(*************************************************************************************2.4Öá¹âÕ¤³ßÎ»ÖÃ¡¢ËÙ¶È¶Ô±È¼ì²é**********************************************************************)
IF  st_Power<>0 THEN
CASE moni_State OF
(*Top Î»ÖÃºÍËÙ¶È±È¶Ô*)
0:
		//实际(*Position*)
		(*Top*)
		Diff_UserTopPos_actual:=ABS(Pos_leftTopLin-Pos_RightTopLin);
		(*Bottom*)
		Diff_UserBottomPos_actual:=ABS(Pos_LeftBottomLin-Pos_RightBottomLin);
		(*Left*)
		Diff_UserLeftPos_actual:=ABS(Pos_LeftTopLin-Pos_LeftBottomLin);
		(*Right*)
		Diff_UserRightPos_actual:=ABS(Pos_RightTopLin-Pos_RightBottomLin);
		(*Velocity*)
		(*Top*)
		Diff_UserTopVelo_actual:=ABS(Velo_leftTopLin-Velo_RightTopLin);
		(*Bottom*)
		Diff_UserBottomVelo_actual:=ABS(Velo_LeftBottomLin-Velo_RightBottomLin);
		(*Left*)
		Diff_UserLeftVelo_actual:=ABS(Velo_LeftTopLin-Velo_LeftBottomLin);
		(*Right*)
		Diff_UserRightVelo_actual:=ABS(Velo_RightTopLin-Velo_RightBottomLin);
		//阈值
		Threshold_UserTopPos_PLC:=Threshold_UserTopPos+UserTaperPositionDisplay;//Top位置误差=gap运动细微误差+目标taper位置
		Threshold_UserTopVelo_PLC:=Threshold_UserTopVelo+ABS(UserGapVelocityDisplay);//Top速度误差=gap运动细微误差+gap目标速度。因为可能出现一个轴运动完了，另一个轴还在运动的情况
		Threshold_UserBottomPos_PLC:=Threshold_UserBottomPos+UserTaperPositionDisplay;//Bottom同上
		Threshold_UserBottomVelo_PLC:=Threshold_UserBottomVelo+ABS(UserGapVelocityDisplay);//Bottom同上
		Threshold_UserLeftPos_PLC:=Threshold_UserLeftPos+UserTaperPositionDisplay;
		Threshold_UserLeftVelo_PLC:=Threshold_UserLeftVelo+ABS(UserGapVelocityDisplay);
		Threshold_UserRightPos_PLC:=Threshold_UserRightPos+UserTaperPositionDisplay;
		Threshold_UserRightVelo_PLC:=Threshold_UserRightVelo+ABS(UserGapVelocityDisplay);
		//比较
		IF Diff_UserTopPos_actual >Threshold_UserTopPos_PLC THEN
				Error:=TRUE;
				ErrorID:=601;
				ErrorDescription:='Diff_UserTopPos_actual >Threshold_UserTopPos_PLC';
				moni_State:=-100;
		ELSIF Diff_UserTopVelo_actual>Threshold_UserTopVelo_PLC  THEN
				Error:=TRUE;
				ErrorID:=602;
				ErrorDescription:='Diff_UserTopVelo_actual>Threshold_UserTopVelo_PLC';
				moni_State:=-100;
		(*Bottom Î»ÖÃºÍËÙ¶È±È¶Ô*)
		ELSIF Diff_UserBottomPos_actual>Threshold_UserBottomPos_PLC THEN
				Error:=TRUE;
				ErrorID:=603;
				ErrorDescription:='Diff_UserBottomPos_actual>Threshold_UserBottomPos_PLC';
				moni_State:=-100;
		ELSIF Diff_UserBottomVelo_actual>Threshold_UserBottomVelo_PLC  THEN
				Error:=TRUE;
				ErrorID:=604;
				ErrorDescription:='Diff_UserBottomVelo_actual>Threshold_UserBottomVelo_PLC';
				moni_State:=-100;
		(*Left Î»ÖÃºÍËÙ¶È±È¶Ô*)
		ELSIF Diff_UserLeftPos_actual>Threshold_UserLeftPos_PLC  THEN
				Error:=TRUE;
				ErrorID:=605;
				ErrorDescription:='Diff_UserLeftPos_actual>Threshold_UserLeftPos_PLC';
				moni_State:=-100;
		ELSIF  Diff_UserLeftVelo_actual>Threshold_UserLeftVelo_PLC THEN
				Error:=TRUE;
				ErrorID:=606;
				ErrorDescription:='Diff_UserLeftVelo_actual>Threshold_UserLeftVelo_PLC';
				moni_State:=-100;
		(*Right Î»ÖÃºÍËÙ¶È±È¶Ô*)
		ELSIF Diff_UserRightPos_actual>Threshold_UserRightPos_PLC  THEN
				Error:=TRUE;
				ErrorID:=607;
				ErrorDescription:='Diff_UserRightPos_actual>Threshold_UserRightPos_PLC';
				moni_State:=-100;
		ELSIF  Diff_UserRightVelo_actual>Threshold_UserRightVelo_PLC THEN
				Error:=TRUE;
				ErrorID:=608;
				ErrorDescription:='Diff_UserRightVelo_actual>Threshold_UserRightVelo_PLC';
				moni_State:=-100;
		END_IF
-100:
		btn_UserGapStop:=TRUE;
		FB_PlcEmergencyStop();
		Error:=TRUE;
		LED_Error:=TRUE;
END_CASE
END_IF
END_ACTION

ACTION A_OneKeyToMaxGap:
//0.上升沿触发
//1.判断电机是否在开启状态,没有就打开电源
//2.判断是否在Moving状态,若有就Stop
//3.将磁间隙打开到至最大阈值
//4.到位后给出反馈
OneKeyToMaxGap_RTRIG(CLK:=btn_OneKeyToMaxGap);
IF OneKeyToMaxGap_RTRIG.Q THEN
	OneKeyToMaxGap_Triggered:=TRUE;
	OneKeyToMaxGap_Done:=FALSE;
END_IF
IF OneKeyToMaxGap_Triggered THEN
	CASE OneKeyToMaxGap_State OF
		0://1.判断电机是否在开启状态,没有就打开电源
			IF st_Power=1 THEN
				OneKeyToMaxGap_State:=1;
			ELSE
				btn_PowerOn:=TRUE;
				IF btn_PowerOn THEN
					A_PowerOn();
				END_IF
			END_IF
		1://1.判断是否在谱学扫描模式，如果是，则切换回正常运动模式
			IF IsSSMotionMode THEN
				SS_Stop:=TRUE;
				IsSSMotionMode:=FALSE;
			END_IF
			OneKeyToMaxGap_State:=2;
		2://判断是否在taper，如果在taper,则判断是否在运动，如果是，则停止运动,0.5sh后，转入下一步
			IF TaperOrNot THEN
				IF moveStatusLeftTop OR moveStatusRightTop OR moveStatusLeftBottom OR moveStatusRightBottom THEN
					btn_UserGapStop:=TRUE;
				ELSE
					OneKeyToMaxGap_TON_Stop2Move_InTaperMode(PT:=T#0.5S);
					OneKeyToMaxGap_TON_Stop2Move_InTaperMode.IN:=TRUE;
					IF OneKeyToMaxGap_TON_Stop2Move_InTaperMode.Q THEN
						TaperOrNot:=FALSE;//关闭taper模式
						OneKeyToMaxGap_State:=3;
						OneKeyToMaxGap_TON_Stop2Move_InTaperMode.IN:=FALSE;
					END_IF
				END_IF
			ELSE
				OneKeyToMaxGap_State:=3;
			END_IF
		3://3.判断是否在Moving状态,若有就Stop.Taper模式已处理完，此处开始走正常GAP开合逻辑
			IF moveStatusLeftTop OR moveStatusRightTop OR moveStatusLeftBottom OR moveStatusRightBottom THEN
				btn_UserGapStop:=TRUE;
			ELSE
				OneKeyToMaxGap_TON_Stop2Move(PT:=T#0.5S);
				OneKeyToMaxGap_TON_Stop2Move.IN:=TRUE;
				IF OneKeyToMaxGap_TON_Stop2Move.Q THEN
					OneKeyToMaxGap_State:=4;
					OneKeyToMaxGap_TON_Stop2Move.IN:=FALSE;
				END_IF
			END_IF
		4://4.将磁间隙打开到至最大阈值
			OneKeyToMaxGap_TON(PT:=INT_TO_TIME(LREAL_TO_INT(max_UserGapPositionNew+30))*1000);
			OneKeyToMaxGap_TON.IN:=TRUE;
			OneKeyToMaxGap_TON_Power2Move(PT:=T#0.1S);
			OneKeyToMaxGap_TON_Power2Move.IN:=TRUE;
			UserGapPositionNew:=max_UserGapPositionNew;
			UserGapVelocityNew:=1;
			btn_UserGapMove:=TRUE;
			IF OneKeyToMaxGap_TON_Power2Move.Q THEN
				OneKeyToMaxGap_TON_Power2Move.IN:=FALSE;
				IF FB_MOVE.BCGapDone THEN
					OneKeyToMaxGap_State:=88;
				END_IF
			END_IF
			IF OneKeyToMaxGap_TON.Q THEN//如果150s后，还没有运动到指定gap，则报错
				OneKeyToMaxGap_TON.IN:=FALSE;
				OneKeyToMaxGap_State:=-100;
			END_IF
		88://6.到位后给出反馈
			OneKeyToMaxGap_Done:=TRUE;	
			Error:=FALSE;
			ErrorID:=0;
			ErrorDescription:='';
			btn_OneKeyToMaxGap:=FALSE;
			OneKeyToMaxGap_Triggered:=FALSE;
			OneKeyToMaxGap_State:=0;
				
		-100:
			OneKeyToMaxGap_Done:=FALSE;
			Error:=TRUE;
			ErrorID:=1705;
			ErrorDescription:='OneKeyToMaxGap Fail';
			btn_OneKeyToMaxGap:=FALSE;
			OneKeyToMaxGap_Triggered:=FALSE;
			OneKeyToMaxGap_State:=0;
	END_CASE
END_IF
END_ACTION

ACTION A_PhaseLowerMotion:
(*输入保护*)
IF btn_UserPhaseLowerMove THEN
	IF NOT inRange_UserPhaseLowerPositionNew THEN
		btn_UserPhaseLowerStop:=TRUE;
		btn_UserPhaseLowerMove:=FALSE;
		Error:=TRUE;
		ErrorId:=812;
		ErrorDescription:='target PhaseLower position out of range,please check';
		RETURN;
	ELSE
		btn_UserPhaseLowerStop:=FALSE;
		Error:=FALSE;
		ErrorId:=0;
		ErrorDescription:='';	
	END_IF
	IF NOT inRange_UserPhaseLowerVelocityNew THEN
		btn_UserPhaseLowerStop:=TRUE;
		btn_UserPhaseLowerMove:=FALSE;
		Error:=TRUE;
		ErrorId:=813;
		ErrorDescription:='target PhaseLower velocity out of range,please check';
		RETURN;
	ELSE
		btn_UserPhaseLowerStop:=FALSE;
		Error:=FALSE;
		ErrorId:=0;
		ErrorDescription:='';
	END_IF
END_IF
(*改变Phase前，先检查Gap，Gap必须处于阈值之上（基本在最大间隙），才能改变Pase*)
IF GapPhase_ChainProtection_On AND UserGapPositionDisplay-GapPhase_ChainProtection_MaxGapValue<-0.01 AND btn_UserPhaseLowerMove THEN
		btn_UserPhaseLowerStop:=TRUE;
		btn_UserPhaseLowerMove:=FALSE;
		Error:=TRUE;
		ErrorId:=814;
		ErrorDescription:='Please Move Gap to MaxGapValue first before move Phase';
		RETURN;
END_IF

(*分别比较四轴目标位置与当前位置的差，如果目标位置比当前位置低，则需要运动到更低-回程差一半；再运动至最终目标位置*)
//只在m=和n=0的时候判断，否则会出现一些BUG，比如往大间隙开时，运动到位后m不能回到0.
IF m_state_PhaseLower=0 AND n_state_PhaseLower=0 THEN
	IF UserPhaseLowerPositionNew-Pos_PhaseLowerLin<-LEDriftErrorThreshold_PhaseLower THEN
			TargetPosLessThanCurrentPos_PhaseLower:=TRUE;
	ELSE
			TargetPosLessThanCurrentPos_PhaseLower:=FALSE;
	END_IF
END_IF

(*Move*)
IF InitPowerDone THEN
		(*目标位置都大于当前位置，直接走到目标位置即可，不需要先走到考虑回城误差的临时位置*)
		IF NOT TargetPosLessThanCurrentPos_PhaseLower AND NOT HysteresisMoving_PhaseLower THEN
			CASE m_state_PhaseLower OF
				0:
					FB_Move_PhaseLower.Mode:=4;						//1.gap;2.single;3.taper;4.debug;5.BCGap&UserMode
					FB_Move_PhaseLower.CoupleState:=st_Couple;			
					FB_Move_PhaseLower.PowerState:=st_Power;							
					FB_Move_PhaseLower.PhaseLowerPosition:=UserPhaseLowerPositionNew;
					FB_Move_PhaseLower.PhaseLowerVelocity:=UserPhaseLowerVelocityNew;		
					IF btn_UserPhaseLowerMove THEN
						FB_Move_PhaseLower.PhaseLowerMove:=TRUE;
						m_state_PhaseLower:=1;
						FB_Move_PhaseLower();
					END_IF
				1:
					btn_UserPhaseLowerMove:=FALSE;
					FB_Move_PhaseLower();
					IF NOT FB_Move_PhaseLower.PhaseLowerDone THEN			(*ÔË¶¯Î´Íê³É£¬Ñ­»·*)
						Led_Run:=TRUE;
						m_state_PhaseLower:=1;
					ELSE									(*ÔË¶¯Íê³É£¬ÏÂÒ»²½*)
						m_state_PhaseLower:=88;
					END_IF
				88:
					btn_UserPhaseLowerMove:=FALSE;					(*×´Ì¬»Ö¸´*)
					Led_Run:=FALSE;
					m_state_PhaseLower:=0;
			END_CASE
		(*四轴有目标位置小于当前位置，先走到临时位置，再走到目标位置*)
		ELSE
			CASE n_state_PhaseLower OF
				0:
					FB_Move_PhaseLower.Mode:=4;						//1.gap;2.single;3.taper;4.debug;5.BCGap&UserMode;5:userMode_2
					FB_Move_PhaseLower.CoupleState:=st_Couple;			
					FB_Move_PhaseLower.PowerState:=st_Power;			
					
					//
					IF TargetPosLessThanCurrentPos_PhaseLower THEN			
						FB_Move_PhaseLower.PhaseLowerPosition:=UserPhaseLowerPositionNew-HysteresisError_PhaseLower;
					ELSE
						FB_Move_PhaseLower.PhaseLowerPosition:=UserPhaseLowerPositionNew;	
					END_IF				
					//
					FB_Move_PhaseLower.PhaseLowerVelocity:=UserPhaseLowerVelocityNew;
						
					IF btn_UserPhaseLowerMove THEN							
						n_state_PhaseLower:=1;
						FB_Move_PhaseLower.PhaseLowerMove:=TRUE;
						FB_Move_PhaseLower();
						HysteresisMoving_PhaseLower:=TRUE;
					END_IF
				1:
					btn_UserPhaseLowerMove:=FALSE;
					FB_Move_PhaseLower();
					IF NOT FB_Move_PhaseLower.PhaseLowerDone THEN			(*还未运动到位置,运动过程中*)
						Led_Run:=TRUE;
						n_state_PhaseLower:=1;
					ELSE									
						n_state_PhaseLower:=2;							(*转到下一步，运动到最终位置*)
						FB_Move_PhaseLower.PhaseLowerMove:=FALSE;
						//Led_Run:=FALSE;
					END_IF
				2:
					FB_Move_PhaseLower.PhaseLowerReset:=FALSE;
					FB_Move_PhaseLower.Mode:=4;						//1.gap;2.single;3.taper;4.debug;5.BCGap&UserMode
					FB_Move_PhaseLower.CoupleState:=st_Couple;			
					FB_Move_PhaseLower.PowerState:=st_Power;			
					FB_Move_PhaseLower.PhaseLowerMove:=TRUE;
					//直接走到目标位置，已经走到位置的，可以继续下命令，只不过它不在走了而已
					FB_Move_PhaseLower.PhaseLowerPosition:=UserPhaseLowerPositionNew;	
					FB_Move_PhaseLower.PhaseLowerVelocity:=UserPhaseLowerVelocityNew;
					FB_Move_PhaseLower();							
					n_state_PhaseLower:=3;
				3:
					FB_Move_PhaseLower();
					IF NOT FB_Move_PhaseLower.PhaseLowerDone THEN			(*还未运动到位置,运动过程中*)
						Led_Run:=TRUE;
						n_state_PhaseLower:=3;
					ELSE									
						n_state_PhaseLower:=88;							(*运动到了最终位置*)
					END_IF
				88:
					btn_UserPhaseLowerMove:=FALSE;					
					Led_Run:=FALSE;
					n_state_PhaseLower:=0;
					HysteresisMoving_PhaseLower:=FALSE;
			END_CASE
		END_IF
	//END_IF
END_IF

IF btn_UserPhaseLowerStop THEN
	FB_Move_PhaseLower.PhaseLowerReset:=TRUE;							(*¸øÔË¶¯FB¸øÍ£Ö¹ÐÅºÅ£¬Ê¹FB_Move×´Ì¬»Ö¸´*)
	FB_Move_PhaseLower();											(*Æô¶¯FB_Move*)
	btn_UserPhaseLowerMove:=FALSE;								(*btn_GapMove:=FALSE*)
	m_state_PhaseLower:=0;	
	n_state_PhaseLower:=0;										(*m_state:=0;*)
	CASE s_state_PhaseLower OF
			0:
				FB_Stop_PhaseLower.Mode:=4;							(*1£ºgapÄ£Ê½£»2£ºµ¥ÁºÄ£Ê½£»3£ºtaperÄ£Ê½£»4£ºDebugÄ£Ê½£»5£ºBCGapÄ£Ê½*)
				FB_Stop_PhaseLower.CoupleState:=st_Couple;			(*ñîºÏ×´Ì¬ÊäÈë*)
				FB_Stop_PhaseLower.PowerState:=st_Power;				(*µçÔ´×´Ì¬ÊäÈë*)
				FB_Stop_PhaseLower.PhaseLowerStop:=TRUE;				(*Execute TRUE*)
				FB_Stop_PhaseLower();								(*Æô¶¯FB*)
				s_state_PhaseLower:=1;
			1:
				FB_Stop_PhaseLower();
				IF NOT FB_Stop_PhaseLower.PhaseLowerDone THEN			(*Í£Ö¹Î´Íê³É£¬Ñ­»·*)
					s_state_PhaseLower:=1;
				ELSE									(*Í£Ö¹Íê³É£¬ÏÂÒ»²½*)
					s_state_PhaseLower:=88;
				END_IF
			88:
				btn_UserPhaseLowerStop:=FALSE;						(*»Ö¸´×´Ì¬*)
				FB_Move_PhaseLower.PhaseLowerReset:=FALSE;				(*ÔËÐÐFB*)
				s_state_PhaseLower:=0;
		END_CASE
END_IF

(*触发限位开关后，相当于点击了Stop按钮*)
FTrig_ReachLS_PhaseLower(CLK:=LS_PhaseLower_Entrance AND LS_PhaseLower_Exit);
IF FTrig_ReachLS_PhaseLower.Q THEN
	btn_UserPhaseLowerStop:=TRUE;
END_IF
END_ACTION

ACTION A_PhaseUpperMotion:
(*输入保护*)
IF btn_UserPhaseUpperMove THEN
	IF NOT inRange_UserPhaseUpperPositionNew THEN
		btn_UserPhaseUpperStop:=TRUE;
		btn_UserPhaseUpperMove:=FALSE;
		Error:=TRUE;
		ErrorId:=809;
		ErrorDescription:='target PhaseUpper position out of range,please check';
		RETURN;
	ELSE
		btn_UserPhaseUpperStop:=FALSE;
		Error:=FALSE;
		ErrorId:=0;
		ErrorDescription:='';	
	END_IF
	IF NOT inRange_UserPhaseUpperVelocityNew THEN
		btn_UserPhaseUpperStop:=TRUE;
		btn_UserPhaseUpperMove:=FALSE;
		Error:=TRUE;
		ErrorId:=810;
		ErrorDescription:='target PhaseUpper velocity out of range,please check';
		RETURN;
	ELSE
		btn_UserPhaseUpperStop:=FALSE;
		Error:=FALSE;
		ErrorId:=0;
		ErrorDescription:='';
	END_IF
END_IF
(*改变Phase前，先检查Gap，Gap必须处于阈值之上（基本在最大间隙），才能改变Pase*)
IF GapPhase_ChainProtection_On AND UserGapPositionDisplay-GapPhase_ChainProtection_MaxGapValue<-0.01 AND btn_UserPhaseUpperMove THEN
		btn_UserPhaseUpperStop:=TRUE;
		btn_UserPhaseUpperMove:=FALSE;
		Error:=TRUE;
		ErrorId:=811;
		ErrorDescription:='Please Move Gap to MaxGapValue first before move Phase';
		RETURN;
END_IF
(*分别比较四轴目标位置与当前位置的差，如果目标位置比当前位置低，则需要运动到更低-回程差一半；再运动至最终目标位置*)
//只在m=和n=0的时候判断，否则会出现一些BUG，比如往大间隙开时，运动到位后m不能回到0.
IF m_state_PhaseUpper=0 AND n_state_PhaseUpper=0 THEN
	IF UserPhaseUpperPositionNew-Pos_PhaseUpperLin<-LEDriftErrorThreshold_PhaseUpper THEN
			TargetPosLessThanCurrentPos_PhaseUpper:=TRUE;
	ELSE
			TargetPosLessThanCurrentPos_PhaseUpper:=FALSE;
	END_IF
END_IF

(*Move*)
IF InitPowerDone THEN
		(*目标位置都大于当前位置，直接走到目标位置即可，不需要先走到考虑回城误差的临时位置*)
		IF NOT TargetPosLessThanCurrentPos_PhaseUpper AND NOT HysteresisMoving_PhaseUpper THEN
			CASE m_state_PhaseUpper OF
				0:
					FB_Move_PhaseUpper.Mode:=4;						//1.gap;2.single;3.taper;4.debug;5.BCGap&UserMode
					FB_Move_PhaseUpper.CoupleState:=st_Couple;			
					FB_Move_PhaseUpper.PowerState:=st_Power;	
					IF btn_UserPhaseUpperMove THEN						
						IF NOT st_Power THEN
							ErrorID:=1501;
							Error:=TRUE;
							ErrorDescription:='Plz PowerOn Frist';
							LED_Error:=TRUE;
							//btn_UserGapMove:=FALSE;
							RETURN;
						ELSE
							ErrorID:=0;
							Error:=FALSE;
							ErrorDescription:='';
							LED_Error:=FALSE;
							//btn_UserGapMove:=TRUE;
						END_IF
						//目标速度位置赋值
						FB_Move_PhaseUpper.PhaseUpperPosition:=UserPhaseUpperPositionNew;
						FB_Move_PhaseUpper.PhaseUpperVelocity:=UserPhaseUpperVelocityNew;		
						//Move
						FB_Move_PhaseUpper.PhaseUpperMove:=TRUE;
						m_state_PhaseUpper:=1;
						FB_Move_PhaseUpper();
					END_IF
				1:
					btn_UserPhaseUpperMove:=FALSE;
					FB_Move_PhaseUpper();
					IF NOT FB_Move_PhaseUpper.PhaseUpperDone THEN			(*ÔË¶¯Î´Íê³É£¬Ñ­»·*)
						Led_Run:=TRUE;
						m_state_PhaseUpper:=1;
					ELSE									(*ÔË¶¯Íê³É£¬ÏÂÒ»²½*)
						m_state_PhaseUpper:=88;
					END_IF
				88:
					btn_UserPhaseUpperMove:=FALSE;					(*×´Ì¬»Ö¸´*)
					Led_Run:=FALSE;
					m_state_PhaseUpper:=0;
			END_CASE
		(*四轴有目标位置小于当前位置，先走到临时位置，再走到目标位置*)
		ELSE
			CASE n_state_PhaseUpper OF
				0:
					FB_Move_PhaseUpper.Mode:=4;						//1.gap;2.single;3.taper;4.debug;5.BCGap&UserMode;5:userMode_2
					FB_Move_PhaseUpper.CoupleState:=st_Couple;			
					FB_Move_PhaseUpper.PowerState:=st_Power;			
					//
					IF btn_UserPhaseUpperMove THEN
						IF NOT st_Power THEN
							ErrorID:=1501;
							Error:=TRUE;
							ErrorDescription:='Plz PowerOn Frist';
							LED_Error:=TRUE;
							//btn_UserGapMove:=FALSE;
							RETURN;
						ELSE
							ErrorID:=0;
							Error:=FALSE;
							ErrorDescription:='';
							LED_Error:=FALSE;
							//btn_UserGapMove:=TRUE;	
						END_IF
						IF TargetPosLessThanCurrentPos_PhaseUpper THEN			
							FB_Move_PhaseUpper.PhaseUpperPosition:=UserPhaseUpperPositionNew-HysteresisError_PhaseUpper;
						ELSE
							FB_Move_PhaseUpper.PhaseUpperPosition:=UserPhaseUpperPositionNew;	
						END_IF				
						//	close gap情况下，加入了PositionNewTemp。//
						//如果在往小间隙运行过程中，改变了目标gap，会在第到达第一次目标位置后，继续向第二
						//次输入的目标运动，而不会回到第一次的目标位置。用temp锁定目标位置
						UserPhaseUpperPositionNewTemp:=UserPhaseUpperPositionNew;
						FB_Move_PhaseUpper.PhaseUpperVelocity:=UserPhaseUpperVelocityNew;
						
						FB_Move_PhaseUpper.PhaseUpperMove:=TRUE;
						FB_Move_PhaseUpper();
						HysteresisMoving_PhaseUpper:=TRUE;
						n_state_PhaseUpper:=1;
					END_IF
				1:
					btn_UserPhaseUpperMove:=FALSE;
					FB_Move_PhaseUpper();
					IF NOT FB_Move_PhaseUpper.PhaseUpperDone THEN			(*还未运动到位置,运动过程中*)
						Led_Run:=TRUE;
						n_state_PhaseUpper:=1;
					ELSE									
						n_state_PhaseUpper:=2;							(*转到下一步，运动到最终位置*)
						FB_Move_PhaseUpper.PhaseUpperMove:=FALSE;
						//Led_Run:=FALSE;
					END_IF
				2:
					FB_Move_PhaseUpper.PhaseUpperReset:=FALSE;
					FB_Move_PhaseUpper.Mode:=4;						//1.gap;2.single;3.taper;4.debug;5.BCGap&UserMode
					FB_Move_PhaseUpper.CoupleState:=st_Couple;			
					FB_Move_PhaseUpper.PowerState:=st_Power;			
					FB_Move_PhaseUpper.PhaseUpperMove:=TRUE;
					//直接走到目标位置，已经走到位置的，可以继续下命令，只不过它不在走了而已
					FB_Move_PhaseUpper.PhaseUpperPosition:=UserPhaseUpperPositionNewTemp;	
					FB_Move_PhaseUpper.PhaseUpperVelocity:=UserPhaseUpperVelocityNew;
					FB_Move_PhaseUpper();							
					n_state_PhaseUpper:=3;
				3:
					FB_Move_PhaseUpper();
					IF NOT FB_Move_PhaseUpper.PhaseUpperDone THEN			(*还未运动到位置,运动过程中*)
						Led_Run:=TRUE;
						n_state_PhaseUpper:=3;
					ELSE									
						n_state_PhaseUpper:=88;							(*运动到了最终位置*)
					END_IF
				88:
					btn_UserPhaseUpperMove:=FALSE;					
					Led_Run:=FALSE;
					n_state_PhaseUpper:=0;
					HysteresisMoving_PhaseUpper:=FALSE;
			END_CASE
		END_IF
	//END_IF
END_IF

IF btn_UserPhaseUpperStop THEN
	FB_Move_PhaseUpper.PhaseUpperReset:=TRUE;							(*¸øÔË¶¯FB¸øÍ£Ö¹ÐÅºÅ£¬Ê¹FB_Move×´Ì¬»Ö¸´*)
	FB_Move_PhaseUpper();											(*Æô¶¯FB_Move*)
	btn_UserPhaseUpperMove:=FALSE;								(*btn_GapMove:=FALSE*)
	m_state_PhaseUpper:=0;	
	n_state_PhaseUpper:=0;										(*m_state:=0;*)
	CASE s_state_PhaseUpper OF
			0:
				FB_Stop_PhaseUpper.Mode:=4;							(*1£ºgapÄ£Ê½£»2£ºµ¥ÁºÄ£Ê½£»3£ºtaperÄ£Ê½£»4£ºDebugÄ£Ê½£»5£ºBCGapÄ£Ê½*)
				FB_Stop_PhaseUpper.CoupleState:=st_Couple;			(*ñîºÏ×´Ì¬ÊäÈë*)
				FB_Stop_PhaseUpper.PowerState:=st_Power;				(*µçÔ´×´Ì¬ÊäÈë*)
				FB_Stop_PhaseUpper.PhaseUpperStop:=TRUE;				(*Execute TRUE*)
				FB_Stop_PhaseUpper();								(*Æô¶¯FB*)
				s_state_PhaseUpper:=1;
			1:
				FB_Stop_PhaseUpper();
				IF NOT FB_Stop_PhaseUpper.PhaseUpperDone THEN			(*Í£Ö¹Î´Íê³É£¬Ñ­»·*)
					s_state_PhaseUpper:=1;
				ELSE									(*Í£Ö¹Íê³É£¬ÏÂÒ»²½*)
					s_state_PhaseUpper:=88;
				END_IF
			88:
				btn_UserPhaseUpperStop:=FALSE;						(*»Ö¸´×´Ì¬*)
				FB_Move_PhaseUpper.PhaseUpperReset:=FALSE;				(*ÔËÐÐFB*)
				s_state_PhaseUpper:=0;
		END_CASE
END_IF

(*触发限位开关后，相当于点击了Stop按钮*)
FTrig_ReachLS_PhaseUpper(CLK:=LS_PhaseUpper_Entrance AND LS_PhaseUpper_Exit);
IF FTrig_ReachLS_PhaseUpper.Q THEN
	btn_UserPhaseUpperStop:=TRUE;
END_IF
END_ACTION

ACTION A_PowerOff:
CASE d_state OF
		0:(*PowerOff*)
			FB_Power(Off:=TRUE);
				d_state:=1;
		1:
			IF NOT FB_power.OffStatus THEN
				d_state:=1;
			ELSE
				d_state:=88;
			END_IF
		88:(*ResetAllState*)
			btn_PowerOn:=FALSE;
			btn_UserGapMove:=FALSE;
			btn_UserGapStop:=FALSE;
			LeftTopLinMoveIndicator:=0;
			RightTopLinMoveIndicator:=0;
			LeftBottomLinMoveIndicator:=0;
			RightBottomLinMoveIndicator:=0;
			fb_ton1.IN:=FALSE;
			fb_ton2.IN:=FALSE;
			fb_ton3.IN:=FALSE;
			State:=0;
			Busy:=FALSE;
			InitPowerDone:=FALSE;
			InitCompensationDatasDone:=FALSE;
			Error:=FALSE;
			ErrorID:=0;
			m_state:=0;
			n_state:=0;
			s_state:=0;
			btn_PowerOff:=FALSE;
			d_state:=0;
			Led_Run:=FALSE;
			Led_Error:=FALSE;
			moni_State:=0;
			i:=0;
END_CASE
END_ACTION

ACTION A_PowerOn:
(****************************************************************
NAME:			A_PowerOn
DATA:			2018.1.9
VERSION:		1.0.0
DESCRIPTION:	
				ÉÏµãÃüÁîºó£¬Ë³ÐòÖ´ÐÐ£º
				1.FB_PowerOn
				·µ»ØÖ´ÐÐÊÇ·ñ³É¹¦
HISTORY:
				2019.1.9		NEW

***************************************************************)
fb_ton3(PT:=t#0.5s);
CASE State OF
	0:	(*FB_Power_On*)
		FB_Power(On:=TRUE);
		fb_ton3.IN:=TRUE;
		State:=1;
	1:	(*wait*)
		FB_power();
		IF NOT FB_power.OnStatus THEN		(*FB_Power_OnÃ»ÓÐÖ´ÐÐÍê£¬wait£¬³¬Ê±FB Error*)
			IF NOT fb_ton3.Q THEN
				State:=1;
			ELSE
				ErrorID:=1;
				State:=99;
			END_IF
		ELSE
			State:=88;
		END_IF
	88:	(*All Done*)
		btn_PowerOn:=FALSE;
		State:=0;
		Error:=FALSE;
		ErrorID:=0;
		Busy:=FALSE;
		InitPowerDone:=TRUE;
		FB_power.On:=FALSE;
		fb_ton3.IN:=FALSE;
		LED_Error:=FALSE;
	99:
		Error:=TRUE;
		//ErrorID:=701;
		//ErrorDescription:='power on error';		
		btn_PowerOn:=FALSE;
		State:=99;
		Busy:=FALSE;
		InitPowerDone:=FALSE;
		fb_ton3.IN:=FALSE;
		LED_Error:=TRUE;
END_CASE
END_ACTION

ACTION A_RegularMotion:
(*如果该ID没有taper需求，则TaperFunctionSolidOn=FALSE，则判定taperOrNot为false*)
IF NOT TaperFunctionSolidOn THEN
	TaperOrNot:=FALSE;
END_IF

(*分别比较四轴目标位置与当前位置的差，如果目标位置比当前位置低，则需要运动到更低-回程差一半；再运动至最终目标位置*)
//只在m=和n=0的时候判断，否则会出现一些BUG，比如往大间隙开时，运动到位后m不能回到0.
IF m_state=0 AND n_state=0 THEN
		TargetPosLessThanCurrentPos:=FALSE;
	IF LeftTopLinPositionNew-Pos_LeftTopLin<-LEDriftErrorThreshold THEN
			TargetPosLessThanCurrentPos:=TRUE;
			TargetLTPosLessThanCurrentLTPos:=TRUE;
	ELSE
				TargetLTPosLessThanCurrentLTPos:=FALSE;
	END_IF
	IF RightTopLinPositionNew-Pos_RightTopLin<-LEDriftErrorThreshold THEN
			TargetPosLessThanCurrentPos:=TRUE;
			TargetRTPosLessThanCurrentRTPos:=TRUE;
	ELSE
			TargetRTPosLessThanCurrentRTPos:=FALSE;
	END_IF
	IF LeftBottomLinPositionNew-Pos_LeftBottomLin<-LEDriftErrorThreshold THEN
			TargetPosLessThanCurrentPos:=TRUE;
			TargetLBPosLessThanCurrentLBPos:=TRUE;
	ELSE
			TargetLBPosLessThanCurrentLBPos:=FALSE;
	END_IF
	IF RightBottomLinPositionNew-Pos_RightBottomLin<-LEDriftErrorThreshold THEN
			TargetPosLessThanCurrentPos:=TRUE;
			TargetRBPosLessThanCurrentRBPos:=TRUE;
	ELSE
			TargetRBPosLessThanCurrentRBPos:=FALSE;
	END_IF
END_IF

(*Move*)
IF InitCompensationDatasDone THEN
		(*四轴目标位置都大于当前位置，直接走到目标位置即可，不需要先走到考虑回城误差的临时位置*)
		IF NOT TargetPosLessThanCurrentPos AND NOT HysteresisMoving THEN
			CASE m_state OF
				0:
					FB_Move.Mode:=5;						//1.gap;2.single;3.taper;4.debug;5.BCGap&UserMode
					FB_Move.CoupleState:=st_Couple;			
					FB_Move.PowerState:=st_Power;						
			
					IF btn_UserGapMove THEN					
						moveStatusGap:=TRUE;
						FB_Move.BCGapReset:=TRUE;
						IF NOT st_Power THEN
							ErrorID:=1501;
							Error:=TRUE;
							ErrorDescription:='Plz PowerOn Frist';
							LED_Error:=TRUE;
							//btn_UserGapMove:=FALSE;
							RETURN;
						ELSE
							ErrorID:=0;
							Error:=FALSE;
							ErrorDescription:='';
							LED_Error:=FALSE;
							//btn_UserGapMove:=TRUE;
						END_IF
						//目标速度位置赋值
						FB_Move.BCLeftTopPosition:=LeftTopLinPositionNew;
						FB_Move.BCRightTopPosition:=RightTopLinPositionNew;
						FB_Move.BCLeftBottomPosition:=LeftBottomLinPositionNew;
						FB_Move.BCRightBottomPosition:=RightBottomLinPositionNew;
						IF NOT TaperOrNot THEN
							FB_Move.BCLeftTopVelocity:=UserGapVelocityNew/2;
							FB_Move.BCRightTopVelocity:=UserGapVelocityNew/2;
							FB_Move.BCLeftBottomVelocity:=UserGapVelocityNew/2;
							FB_Move.BCRightBottomVelocity:=UserGapVelocityNew/2;
						ELSE
							FB_Move.BCLeftTopVelocity:=UserTaperVelocityNew;
							FB_Move.BCRightTopVelocity:=UserTaperVelocityNew;
							FB_Move.BCLeftBottomVelocity:=UserTaperVelocityNew;
							FB_Move.BCRightBottomVelocity:=UserTaperVelocityNew;
						END_IF
						m_state:=1;
						FB_Move();
					END_IF
				1:
					FB_Move.BCGapMove:=TRUE;
					btn_UserGapMove:=FALSE;
					FB_Move();
					IF NOT FB_Move.BCGapDone THEN			(*ÔË¶¯Î´Íê³É£¬Ñ­»·*)
						Led_Run:=TRUE;
						m_state:=1;
					ELSE									(*ÔË¶¯Íê³É£¬ÏÂÒ»²½*)
						m_state:=88;
					END_IF
				88:
					moveStatusGap:=FALSE;
					btn_UserGapMove:=FALSE;					(*×´Ì¬»Ö¸´*)
					Led_Run:=FALSE;
					m_state:=0;
			END_CASE
		(*四轴有目标位置小于当前位置，先走到临时位置，再走到目标位置*)
		ELSE
			CASE n_state OF
				0:
					FB_Move.Mode:=5;						//1.gap;2.single;3.taper;4.debug;5.BCGap&UserMode;5:userMode_2
					FB_Move.CoupleState:=st_Couple;			
					FB_Move.PowerState:=st_Power;			
					IF btn_UserGapMove THEN	
						FB_Move.BCGapReset:=TRUE;					
						moveStatusGap:=TRUE;
						IF NOT st_Power THEN
							ErrorID:=1501;
							Error:=TRUE;
							ErrorDescription:='Plz PowerOn Frist';
							LED_Error:=TRUE;
							//btn_UserGapMove:=FALSE;
							RETURN;
						ELSE
							ErrorID:=0;
							Error:=FALSE;
							ErrorDescription:='';
							LED_Error:=FALSE;
							//btn_UserGapMove:=TRUE;
						END_IF						
						//
						IF TargetLTPosLessThanCurrentLTPos THEN			
							FB_Move.BCLeftTopPosition:=LeftTopLinPositionNew-HysteresisError/2;
						ELSE
							FB_Move.BCLeftTopPosition:=LeftTopLinPositionNew;	
						END_IF
						//
						IF TargetRTPosLessThanCurrentRTPos THEN 
							FB_Move.BCRightTopPosition:=RightTopLinPositionNew-HysteresisError/2;
						ELSE					
							FB_Move.BCRightTopPosition:=RightTopLinPositionNew;
						END_IF
						//
						IF TargetLBPosLessThanCurrentLBPos THEN
							FB_Move.BCLeftBottomPosition:=LeftBottomLinPositionNew-HysteresisError/2;
						ELSE
							FB_Move.BCLeftBottomPosition:=LeftBottomLinPositionNew;
						END_IF
						//
						IF TargetRBPosLessThanCurrentRBPos THEN
							FB_Move.BCRightBottomPosition:=RightBottomLinPositionNew-HysteresisError/2;
						ELSE
							FB_Move.BCRightBottomPosition:=RightBottomLinPositionNew;
						END_IF	
						//	close gap情况下，加入了LeftTopLinPositionNewTemp。//
						//如果在往小间隙运行过程中，改变了目标gap，会在第到达第一次目标位置后，继续向第二
						//次输入的目标运动，而不会回到第一次的目标位置。用temp锁定目标位置
						LeftTopLinPositionNewTemp:=LeftTopLinPositionNew;
						RightTopLinPositionNewTemp:=RightTopLinPositionNew;
						LeftBottomLinPositionNewTemp:=LeftBottomLinPositionNew;
						RightBottomLinPositionNewTemp:=RightBottomLinPositionNew;
			
						//
						IF NOT TaperOrNot THEN
							FB_Move.BCLeftTopVelocity:=UserGapVelocityNew/2;
							FB_Move.BCRightTopVelocity:=UserGapVelocityNew/2;
							FB_Move.BCLeftBottomVelocity:=UserGapVelocityNew/2;
							FB_Move.BCRightBottomVelocity:=UserGapVelocityNew/2;
							IF UserGapVelocityNew >1 THEN								  
								ErrorID:=1502;
								Error:=TRUE;
								ErrorDescription:='UserGapVelocityNew must<=1';
								LED_Error:=TRUE;
								btn_UserGapMove:=FALSE;
								RETURN;
							ELSE
								ErrorID:=0;
								Error:=FALSE;
								ErrorDescription:='';
								LED_Error:=FALSE;	
							END_IF									
						ELSE
							FB_Move.BCLeftTopVelocity:=UserTaperVelocityNew;
							FB_Move.BCRightTopVelocity:=UserTaperVelocityNew;
							FB_Move.BCLeftBottomVelocity:=UserTaperVelocityNew;
							FB_Move.BCRightBottomVelocity:=UserTaperVelocityNew;
						END_IF	

						FB_Move();
						HysteresisMoving:=TRUE;		
						n_state:=1;	
					END_IF
				1:
					btn_UserGapMove:=FALSE;	
					FB_Move.BCGapMove:=TRUE;
					FB_Move();
					IF NOT FB_Move.BCGapDone THEN			(*还未运动到位置,运动过程中*)
						Led_Run:=TRUE;
						n_state:=1;
					ELSE									
						n_state:=2;							(*转到下一步，运动到最终位置*)
						FB_Move.BCGapMove:=FALSE;
						//Led_Run:=FALSE;
					END_IF
				2:
					FB_Move.BCGapReset:=FALSE;
					FB_Move.Mode:=5;						//1.gap;2.single;3.taper;4.debug;5.BCGap&UserMode
					FB_Move.CoupleState:=st_Couple;			
					FB_Move.PowerState:=st_Power;			
					FB_Move.BCGapMove:=TRUE;
					//直接走到目标位置，已经走到位置的，可以继续下命令，只不过它不在走了而已
					FB_Move.BCLeftTopPosition:=LeftTopLinPositionNewTemp;	
					FB_Move.BCRightTopPosition:=RightTopLinPositionNewTemp;
					FB_Move.BCLeftBottomPosition:=LeftBottomLinPositionNewTemp;
					FB_Move.BCRightBottomPosition:=RightBottomLinPositionNewTemp;
					//
					IF NOT TaperOrNot THEN
						FB_Move.BCLeftTopVelocity:=UserGapVelocityNew/2;
						FB_Move.BCRightTopVelocity:=UserGapVelocityNew/2;
						FB_Move.BCLeftBottomVelocity:=UserGapVelocityNew/2;
						FB_Move.BCRightBottomVelocity:=UserGapVelocityNew/2;
					ELSE
						FB_Move.BCLeftTopVelocity:=UserTaperVelocityNew;
						FB_Move.BCRightTopVelocity:=UserTaperVelocityNew;
						FB_Move.BCLeftBottomVelocity:=UserTaperVelocityNew;
						FB_Move.BCRightBottomVelocity:=UserTaperVelocityNew;
					END_IF
					FB_Move();							
					n_state:=3;
				3:
					FB_Move();
					IF NOT FB_Move.BCGapDone THEN			(*还未运动到位置,运动过程中*)
						Led_Run:=TRUE;
						n_state:=3;
					ELSE									
						n_state:=88;							(*运动到了最终位置*)
					END_IF
					(*
					IF NOT Unreach_LS_Bottom THEN
						n_state:=88;							(*在运动过程中如果碰到下限位，则也转到下一步，运动到最终位置*)
						FB_Move.BCGapMove_2:=FALSE;
					END_IF
					*)
				88:				
					moveStatusGap:=FALSE;
					btn_UserGapMove:=FALSE;					
					Led_Run:=FALSE;
					n_state:=0;
					HysteresisMoving:=FALSE;
			END_CASE
		END_IF
	//
	//FB_Move.BCLeftTopPosition等四轴位置监控
	//
END_IF

//
//STOP
//
CASE s_state OF
	0:
		IF btn_UserGapStop OR btn_Reset THEN					
			moveStatusGap:=FALSE;
			m_state:=0;	
			n_state:=0;	
			HysteresisMoving:=FALSE;
					
			FB_Stop.Mode:=5;	
			FB_Stop.CoupleState:=st_Couple;	
			FB_Stop.PowerState:=st_Power;
			FB_Stop.BCGapStop:=TRUE;
			FB_Stop();	
			s_state:=1;
		END_IF
	1:
		btn_UserGapStop:=FALSE;	
		FB_Stop();
		IF NOT FB_Stop.BCGapDone THEN
			s_state:=1;
		ELSE
			s_state:=88;
		END_IF
	88:
		FB_Move.BCGapReset:=FALSE;
		btn_reset:=FALSE;
		s_state:=0;
END_CASE

(*触发限位开关后，相当于点击了Stop按钮*)
FTrig_ReachLS(CLK:=Unreach_LS_Far AND Unreach_LS_Near);
IF FTrig_ReachLS.Q THEN
	btn_UserGapStop:=TRUE;
END_IF
(*触发限位后，如果继续向前运动，点击move，则相当于点击stop，用于恢复move的状态位*)
IF NOT Unreach_LS_Far AND btn_UserGapMove AND UserGapPositionNew >= UserGapPositionDisplay THEN
	btn_UserGapStop:=TRUE;
END_IF
IF NOT Unreach_LS_Near AND btn_UserGapMove AND UserGapPositionNew <= UserGapPositionDisplay THEN
	btn_UserGapStop:=TRUE;
END_IF
END_ACTION

ACTION A_SpectroscopyScanningMotion:
(*输入保护*)
IF SS_Move AND SSMotionMode AND NOT RegularMotionMode THEN
	IF NOT inRange_SS_StepSize THEN
		SS_Stop:=TRUE;
		SS_Move:=FALSE;
		Error:=TRUE;
		ErrorId:=805;
		ErrorDescription:='target StepSize out of range,please check';
		RETURN;
	ELSE
		//SS_Stop:=FALSE;
		Error:=FALSE;
		ErrorId:=0;
		ErrorDescription:='';	
	END_IF
	//
	IF NOT inRange_SS_StepNumber THEN
		SS_Stop:=TRUE;
		SS_Move:=FALSE;
		Error:=TRUE;
		ErrorId:=806;
		ErrorDescription:='target StepNumber out of range,please check';
		RETURN;
	ELSE
		//SS_Stop:=FALSE;
		Error:=FALSE;
		ErrorId:=0;
		ErrorDescription:='';	
	END_IF
	IF NOT inRange_SS_StepVelocity THEN
		SS_Stop:=TRUE;
		SS_Move:=FALSE;
		Error:=TRUE;
		ErrorId:=807;
		ErrorDescription:='target StepVelocity out of range,please check';
		RETURN;
	ELSE
		//SS_Stop:=FALSE;
		Error:=FALSE;
		ErrorId:=0;
		ErrorDescription:='';	
	END_IF
	IF NOT inRange_StepEachTime_ms THEN
		SS_Stop:=TRUE;
		SS_Move:=FALSE;
		Error:=TRUE;
		ErrorId:=808;
		ErrorDescription:='target StepEachTime_ms out of range,please check';
		RETURN;
	ELSE
		//SS_Stop:=FALSE;
		Error:=FALSE;
		ErrorId:=0;
		ErrorDescription:='';	
	END_IF
END_IF
(*单步时长转换*)
StepEachTime:=INT_TO_TIME(StepEachTime_ms);
SS_TON(PT:=StepEachTime);
(*上升沿触发，初始SS位置=当前磁间隙*)
RTRG_SS_StartPositionDisplay(CLK:=SS_Move);
IF RTRG_SS_StartPositionDisplay.Q THEN
	SS_StartPositionDisplay:=UserGapPositionDisplay;
	SS_InitStartPositionDone:=TRUE;
END_IF
(*SS主程序*)
IF InitPowerDone AND InitCompensationDatasDone AND SS_Move AND SS_InitStartPositionDone THEN
	IF NOT st_Power THEN
		ErrorID:=1501;
		Error:=TRUE;
		ErrorDescription:='Plz PowerOn Frist';
		LED_Error:=TRUE;
		//btn_UserGapMove:=FALSE;
		RETURN;
	ELSE
		ErrorID:=0;
		Error:=FALSE;
		ErrorDescription:='';
		LED_Error:=FALSE;
		//btn_UserGapMove:=TRUE;
	END_IF	
CASE SS_MoveState OF
		0:
				//UserGapPositionNew:=UserGapPositionDisplay+SS_StepSize;
				UserGapPositionNew:=SS_StartPositionDisplay+SS_StepSize*(SS_currentStep+1);
				A_InitCompensationData();
				FB_Move.Mode:=5;						//1.gap;2.single;3.taper;4.debug;5.BCGap&UserMode
				FB_Move.CoupleState:=st_Couple;			
				FB_Move.PowerState:=st_Power;							
				FB_Move.BCLeftTopPosition:=LeftTopLinPositionNew;
				FB_Move.BCLeftTopVelocity:=SS_StepVelocity/2;
				FB_Move.BCRightTopPosition:=RightTopLinPositionNew;
				FB_Move.BCRightTopVelocity:=SS_StepVelocity/2;
				FB_Move.BCLeftBottomPosition:=LeftBottomLinPositionNew;
				FB_Move.BCLeftBottomVelocity:=SS_StepVelocity/2;
				FB_Move.BCRightBottomPosition:=RightBottomLinPositionNew;
				FB_Move.BCRightBottomVelocity:=SS_StepVelocity/2;		
				FB_Move.BCGapMove:=TRUE;
				FB_Move();
				SS_MoveState:=1;
		1:
				SS_TON.IN:=TRUE;
				FB_Move();
				IF FB_Move.GapMoving AND NOT SS_TimeCountBegin THEN
					SS_StepSystemTime_Begin[SS_currentStep]:=F_GetSysTime();
					SS_TimeCountBegin:=TRUE;
				END_IF
				IF NOT FB_Move.BCGapDone THEN			
					Led_Run:=TRUE;
					SS_MoveState:=1;
				ELSE									
					SS_MoveState:=66;
					SS_StepSystemTime_End[SS_currentStep]:=F_GetSysTime();
					SS_StepCountTime[SS_currentStep]:=SS_StepSystemTime_End[SS_currentStep]-SS_StepSystemTime_Begin[SS_currentStep];
					SS_TimeCountBegin:=FALSE;
				END_IF
		66:
				SS_currentStep:=SS_currentStep+1;			
				Led_Run:=FALSE;
				IF SS_currentStep=SS_StepNumber THEN								
					SS_MoveState:=88;
				END_IF
				IF SS_currentStep<SS_StepNumber THEN
					SS_MoveState:=77;
				END_IF
		77://等待单步时长够
				IF SS_TON.Q THEN
					SS_TON.IN:=FALSE;
					SS_MoveState:=0;
				END_IF
		88:
				SS_TON.IN:=FALSE;
				SS_Move:=FALSE;	
				Led_Run:=FALSE;
				SS_MoveState:=0;
				SS_currentStep:=0;
				SS_InitStartPositionDone:=FALSE;
				//SS_StepSystemTime[SS_StepNumber]:=F_GetSysTime();
	END_CASE
END_IF
(*获取每一步耗时*)
//FOR	m:= 0 TO SS_StepNumber DO
//	SS_StepCountTime[m]:=(SS_StepSystemTime_End[m]-SS_StepSystemTime_Begin[m]);
//END_FOR

(*STOP*)
IF SS_Stop OR btn_reset THEN
	FB_Move.BCGapReset:=TRUE;							(*¸øÔË¶¯FB¸øÍ£Ö¹ÐÅºÅ£¬Ê¹FB_Move×´Ì¬»Ö¸´*)
	FB_Move();											(*Æô¶¯FB_Move*)
	SS_Move:=FALSE;								(*btn_GapMove:=FALSE*)
	SS_MoveState:=0;										(*m_state:=0;*)
	CASE SS_StopState OF
			0:
				FB_Stop.Mode:=5;							(*1£ºgapÄ£Ê½£»2£ºµ¥ÁºÄ£Ê½£»3£ºtaperÄ£Ê½£»4£ºDebugÄ£Ê½£»5£ºBCGapÄ£Ê½*)
				FB_Stop.CoupleState:=st_Couple;			(*ñîºÏ×´Ì¬ÊäÈë*)
				FB_Stop.PowerState:=st_Power;				(*µçÔ´×´Ì¬ÊäÈë*)
				FB_Stop.BCGapStop:=TRUE;				(*Execute TRUE*)
				FB_Stop();								(*Æô¶¯FB*)
				SS_StopState:=1;
			1:
				FB_Stop();
				IF NOT FB_Stop.BCGapDone THEN			(*Í£Ö¹Î´Íê³É£¬Ñ­»·*)
					SS_StopState:=1;
				ELSE									(*Í£Ö¹Íê³É£¬ÏÂÒ»²½*)
					SS_StopState:=88;
				END_IF
			88:
				SS_Stop:=FALSE;						(*»Ö¸´×´Ì¬*)
				FB_Move.BCGapReset:=FALSE;				(*ÔËÐÐFB*)
				SS_StopState:=0;
				btn_reset:=FALSE;
				//SS_Stop2:=FALSE;
		END_CASE
END_IF

(*触发限位开关后，相当于点击了Stop按钮*)
FTrig_ReachLS(CLK:=Unreach_LS_Far AND Unreach_LS_Near);
IF FTrig_ReachLS.Q THEN
	SS_Stop:=TRUE;
END_IF
END_ACTION

END_PROGRAM

// ---- POUs/TiltSensor/SAFE.TcPOU
PROGRAM SAFE
VAR
	TiltSensorFunctionOn:BOOL;
	//
	//Top TiltSensor
	//
	TiltSensorTopAngle_INT AT%I*: INT;
	TiltSensorTopAngle_mA: LREAL;
	TileSensorTop_SN:STRING:='TT1026';
	TiltSensorTop_ScaleFactor: LREAL:=0.201;
	fbMovingAvg_TiltSensorTop : FB_Simple_MovingAvg;
	TiltSensorTop_FilterWindow : INT := 1000;  // 100个周期平均 = 1000ms
	TiltSensorTop_mA_Filter:LREAL;
	TiltSensorTop_mA:LREAL;
	//角度，单位：°
	TiltSensorTopAngle: LREAL;	
	//滤波后角度，单位：°
	TiltSensorTopAngle_Filter: LREAL;
	TileSensorTop_Underrange AT%I*:BOOL;
	TileSensorTop_Overrange AT%I*:BOOL;
	TileSensorTop_Error AT%I*:BOOL;
	TiltSensorTopAngle_mA_Filter: LREAL;
	//TileMotorOffset: REAL;
	//L_Center2Motor: INT:=1375;
	//初始准直零位角度
	TiltSensorTop_InitAngle:LREAL;
	//角度阈值
	TiltSensorTop_GapThreshold:LREAL;
	TiltSensorTop_IDTaperThreshold:LREAL;
	TiltSensorTop_BLTaperThreshold:LREAL;
	TiltSensorTop_SingleCarrierThreshold:LREAL;
	TiltSensorTop_DebugThreshold:LREAL;
	//角度与taper的比例
	TaperAndTileTopAngleScale:LREAL;
		//
	//Bottom TiltSensor
	//
	TiltSensorBottomAngle_INT AT%I*: INT;
	TiltSensorBottomAngle_mA: LREAL;
	TileSensorBottom_SN:STRING:='TT1026';
	TiltSensorBottom_ScaleFactor: LREAL:=0.0596;
	fbMovingAvg_TiltSensorBottom : FB_Simple_MovingAvg;
	TiltSensorBottom_FilterWindow : INT := 1000;  // 100个周期平均 = 1000ms
	TiltSensorBottom_mA_Filter:LREAL;
	TiltSensorBottom_mA:LREAL;
	//角度，单位：°
	TiltSensorBottomAngle: LREAL;	
	//滤波后角度，单位：°
	TiltSensorBottomAngle_Filter: LREAL;
	TileSensorBottom_Underrange AT%I*:BOOL;
	TileSensorBottom_Overrange AT%I*:BOOL;
	TileSensorBottom_Error AT%I*:BOOL;
	TiltSensorBottomAngle_mA_Filter: LREAL;
	//TileMotorOffset: REAL;
	//L_Center2Motor: INT:=1375;
	//初始准直零位角度
	TiltSensorBottom_InitAngle:LREAL;
	//角度阈值
	TiltSensorBottom_GapThreshold:LREAL;
	TiltSensorBottom_IDTaperThreshold:LREAL;
	TiltSensorBottom_BLTaperThreshold:LREAL;
	TiltSensorBottom_SingleCarrierThreshold:LREAL;
	TiltSensorBottom_DebugThreshold:LREAL;
	//角度与taper的比例
	TaperAndTileBottomAngleScale:LREAL;
	
	a: LREAL;
END_VAR

//
//Function On/OFF
//
IF NOT TiltSensorFunctionOn THEN
	RETURN;
END_IF
//
//Top TiltSensor
//
TiltSensorTopAngle_mA:=(INT_TO_LREAL(TiltSensorTopAngle_INT)/32767)*16+4;
// 每个PLC周期（10ms）调用一次,移动平均
fbMovingAvg_TiltSensorTop(x := TiltSensorTopAngle_mA,    // 输入原始值
            N := TiltSensorTop_FilterWindow,  // 窗口大小
            rst := FALSE,       // 不复位
            y => TiltSensorTopAngle_mA_Filter);     // 输出平均值
//计算角度
TiltSensorTopAngle_Filter:=DINT_TO_LREAL(LREAL_TO_DINT(((TiltSensorTopAngle_mA_Filter-12)*(TiltSensorTop_ScaleFactor)+TiltSensorTop_InitAngle)*100000))/100000;//滤波后
TiltSensorTopAngle:=DINT_TO_LREAL(LREAL_TO_DINT(((TiltSensorTopAngle_mA-12)*(TiltSensorTop_ScaleFactor)+TiltSensorTop_InitAngle)*100000))/100000;//未滤波，原始数据
//计算电机处由于倾斜导致的偏移量，单位毫米
//TileMotorOffset:=L_Center2Motor*2*TAN(TiltSensorAngle_degree*PI / 180);
//阈值触发
(*先分几种大梁运动模式，每种模式再细分*)
IF MAIN.pbUserMode THEN
	IF NormalGapMode THEN
		IF TiltSensorTopAngle>TiltSensorTop_GapThreshold THEN
			ErrorID:=1601;
			Error:=TRUE;
			ErrorDescription:='TiltSensorTopAngle>TiltSensorTop_Threshold';
			FB_PlcEmergencyStop();
			LED_Error:=TRUE;
		END_IF
	END_IF
	IF IDTaperMode THEN
		IF TiltSensorTopAngle>TiltSensorTop_IDTaperThreshold THEN
			ErrorID:=1602;
			Error:=TRUE;
			ErrorDescription:='TiltSensorTopAngle>TiltSensorTop_IDTaperThreshold';
			FB_PlcEmergencyStop();
			LED_Error:=TRUE;
		END_IF
	END_IF
	IF BLTaperMode THEN
		IF TiltSensorTopAngle>TiltSensorTop_BLTaperThreshold THEN
			ErrorID:=1603;
			Error:=TRUE;
			ErrorDescription:='TiltSensorTopAngle>TiltSensorTop_BLTaperThreshold';
			FB_PlcEmergencyStop();
			LED_Error:=TRUE;
		END_IF
	END_IF
ELSIF MAIN.pbSingleCarrierMode THEN
	IF TiltSensorTopAngle>TiltSensorTop_SingleCarrierThreshold THEN
		ErrorID:=1604;
		Error:=TRUE;
		ErrorDescription:='TiltSensorTopAngle>TiltSensorTop_SingleCarrierThreshold';
		FB_PlcEmergencyStop();
		LED_Error:=TRUE;
	END_IF
ELSIF MAIN.pbDebugMode THEN
	IF TiltSensorTopAngle>TiltSensorTop_DebugThreshold THEN
		ErrorID:=1605;
		Error:=TRUE;
		ErrorDescription:='TiltSensorTopAngle>TiltSensorTop_DebugThreshold';
		FB_PlcEmergencyStop();
		LED_Error:=TRUE;
	END_IF
END_IF
//角度与taper的比例
IF NormalGapMode THEN
	TaperAndTileTopAngleScale:=0;
ELSIF IDTaperMode THEN
	TaperAndTileTopAngleScale:=DINT_TO_LREAL(LREAL_TO_DINT((ATAN((UserMode.UserTaperPositionNew/2)/(2*UserMode.L_Center2Motor))*180/PI)*100000))/100000;
ELSIF BLTaperMode THEN
	TaperAndTileTopAngleScale:=DINT_TO_LREAL(LREAL_TO_DINT((ATAN((UserMode.BLUserTaperPositionNew/4)/(UserMode.L_HalfGirder))*180/PI)*100000))/100000;
END_IF
(*
//超出检测范围处理
IF TileSensorTop_Underrange THEN
	ErrorID:=1604;
	Error:=TRUE;
	ErrorDescription:='TileSensorTop_Underrange';
	//FB_PlcEmergencyStop();
	LED_Error:=TRUE;
ELSE
	ErrorID:=0;
	Error:=FALSE;
	ErrorDescription:='';
	LED_Error:=FALSE;
END_IF
IF TileSensorTop_Overrange THEN
	ErrorID:=1605;
	Error:=TRUE;
	ErrorDescription:='TileSensorTop_Overrange';
	//FB_PlcEmergencyStop();
	LED_Error:=TRUE;
ELSE
	ErrorID:=0;
	Error:=FALSE;
	ErrorDescription:='';
	LED_Error:=FALSE;
END_IF
IF TileSensorTop_Error THEN
	ErrorID:=1606;
	Error:=TRUE;
	ErrorDescription:='TileSensorTop_Error';
	//FB_PlcEmergencyStop();
	LED_Error:=TRUE;
ELSE
	ErrorID:=0;
	Error:=FALSE;
	ErrorDescription:='';
	LED_Error:=FALSE;
END_IF
*)
//
//Bottom TiltSensor
//
TiltSensorBottomAngle_mA:=(INT_TO_LREAL(TiltSensorBottomAngle_INT)/32767)*16+4;
// 每个PLC周期（10ms）调用一次,移动平均
fbMovingAvg_TiltSensorBottom(x := TiltSensorBottomAngle_mA,    // 输入原始值
            N := TiltSensorBottom_FilterWindow,  // 窗口大小
            rst := FALSE,       // 不复位
            y => TiltSensorBottomAngle_mA_Filter);     // 输出平均值
//计算角度
TiltSensorBottomAngle_Filter:=DINT_TO_LREAL(LREAL_TO_DINT(((TiltSensorBottomAngle_mA_Filter-12)*TiltSensorBottom_ScaleFactor+TiltSensorBottom_InitAngle)*100000))/100000;//滤波后
TiltSensorBottomAngle:=DINT_TO_LREAL(LREAL_TO_DINT(((TiltSensorBottomAngle_mA-12)*TiltSensorBottom_ScaleFactor+TiltSensorBottom_InitAngle)*100000))/100000;//未滤波，原始数据
//计算电机处由于倾斜导致的偏移量，单位毫米
//TileMotorOffset:=L_Center2Motor*2*TAN(TiltSensorAngle_degree*PI / 180);
//阈值触发
IF MAIN.pbUserMode THEN
	IF NormalGapMode THEN
		IF TiltSensorBottomAngle>TiltSensorBottom_GapThreshold THEN
			ErrorID:=1606;
			Error:=TRUE;
			ErrorDescription:='TiltSensorBottomAngle>TiltSensorBottom_Threshold';
			FB_PlcEmergencyStop();
			LED_Error:=TRUE;
		END_IF
	END_IF
	IF IDTaperMode THEN
		IF TiltSensorBottomAngle>TiltSensorBottom_IDTaperThreshold THEN
			ErrorID:=1607;
			Error:=TRUE;
			ErrorDescription:='TiltSensorBottomAngle>TiltSensorBottom_IDTaperThreshold';
			FB_PlcEmergencyStop();
			LED_Error:=TRUE;
		END_IF
	END_IF
	IF BLTaperMode THEN
		IF TiltSensorBottomAngle>TiltSensorBottom_BLTaperThreshold THEN
			ErrorID:=1608;
			Error:=TRUE;
			ErrorDescription:='TiltSensorBottomAngle>TiltSensorBottom_BLTaperThreshold';
			FB_PlcEmergencyStop();
			LED_Error:=TRUE;
		END_IF
	END_IF
ELSIF MAIN.pbSingleCarrierMode THEN
	IF TiltSensorBottomAngle>TiltSensorBottom_SingleCarrierThreshold THEN
		ErrorID:=1609;
		Error:=TRUE;
		ErrorDescription:='TiltSensorTopAngle>TiltSensorBottom_SingleCarrierThreshold';
		FB_PlcEmergencyStop();
		LED_Error:=TRUE;
	END_IF
ELSIF MAIN.pbDebugMode THEN
	IF TiltSensorBottomAngle>TiltSensorBottom_DebugThreshold THEN
		ErrorID:=1610;
		Error:=TRUE;
		ErrorDescription:='TiltSensorBottomAngle>TiltSensorBottom_DebugThreshold';
		FB_PlcEmergencyStop();
		LED_Error:=TRUE;
	END_IF
END_IF
//角度与taper的比例
IF NormalGapMode THEN
	TaperAndTileBottomAngleScale:=0;
ELSIF IDTaperMode THEN
	TaperAndTileBottomAngleScale:=DINT_TO_LREAL(LREAL_TO_DINT((ATAN((UserMode.UserTaperPositionNew/2)/(2*UserMode.L_Center2Motor))*180/PI)*100000))/100000;;
ELSIF BLTaperMode THEN
	TaperAndTileBottomAngleScale:=DINT_TO_LREAL(LREAL_TO_DINT((ATAN((UserMode.BLUserTaperPositionNew/4)/(UserMode.L_HalfGirder))*180/PI)*100000))/100000;;
END_IF
(*
//超出检测范围处理
IF TileSensorBottom_Underrange THEN
	ErrorID:=1610;
	Error:=TRUE;
	ErrorDescription:='TileSensorBottom_Underrange';
	//FB_PlcEmergencyStop();
	LED_Error:=TRUE;
ELSE
	ErrorID:=0;
	Error:=FALSE;
	ErrorDescription:='';
	LED_Error:=FALSE;
END_IF
IF TileSensorBottom_Overrange THEN
	ErrorID:=1611;
	Error:=TRUE;
	ErrorDescription:='TileSensorBottom_Overrange';
	//FB_PlcEmergencyStop();
	LED_Error:=TRUE;
ELSE
	ErrorID:=0;
	Error:=FALSE;
	ErrorDescription:='';
	LED_Error:=FALSE;
END_IF
IF TileSensorBottom_Error THEN
	ErrorID:=1612;
	Error:=TRUE;
	ErrorDescription:='TileSensorBottom_Error';
	//FB_PlcEmergencyStop();
	LED_Error:=TRUE;
ELSE
	ErrorID:=0;
	Error:=FALSE;
	ErrorDescription:='';
	LED_Error:=FALSE;
END_IF
*)

END_PROGRAM
